FUNCTION_BLOCK MagneticGripper (* Composite FB wrapping other FBs *)
  (* Standard: 61499-2 *)
  (* Version 1.0, 2021-03-18, AK120569 *)
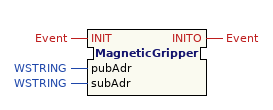
  EVENT_INPUT
    INIT; (* Initialization Request *)
  END_EVENT
  EVENT_OUTPUT
    INITO; (* Initialization Confirm *)
  END_EVENT
  VAR_INPUT
    pubAdr : WSTRING;
    subAdr : WSTRING;
  END_VAR
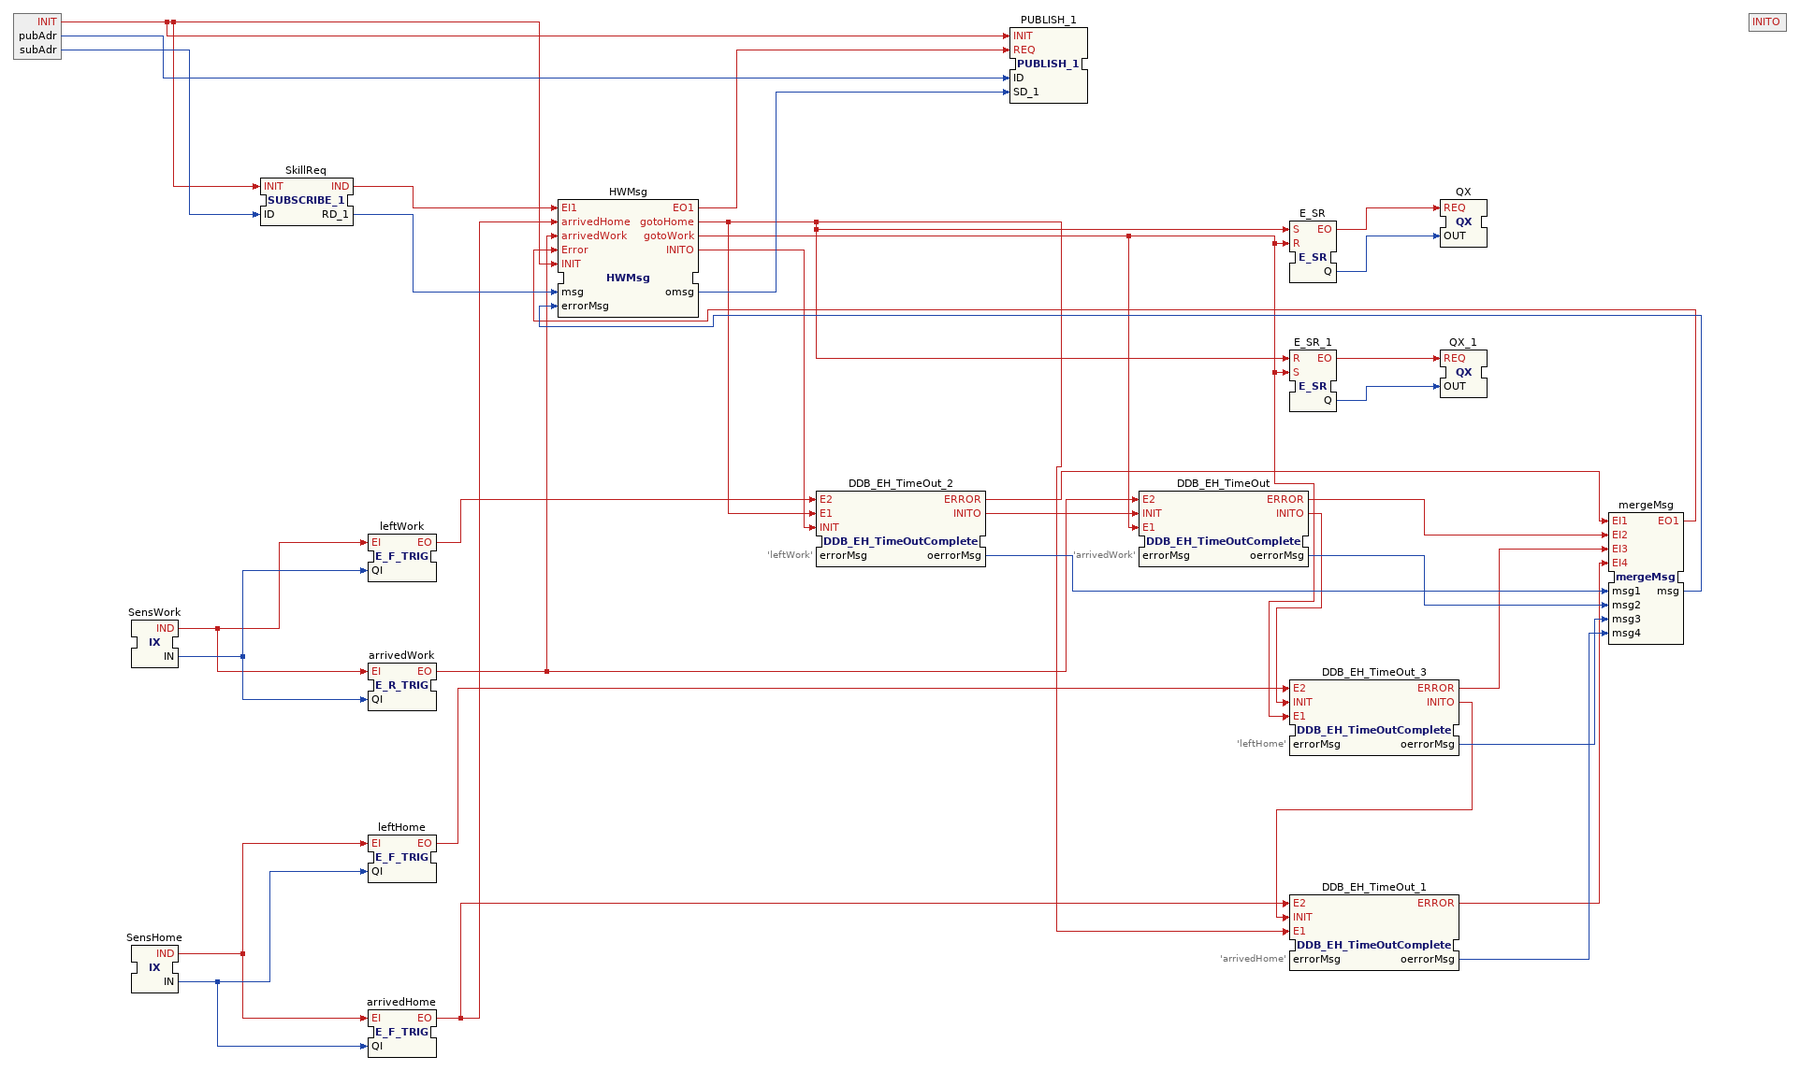
  FBS
    SkillReq : SUBSCRIBE_1;
    SensHome : IX;
    SensWork : IX;
    arrivedHome : E_F_TRIG;
    arrivedWork : E_R_TRIG;
    DDB_EH_TimeOut_1 : DDB_EH_TimeOutComplete(errorMsg := 'arrivedHome');
    DDB_EH_TimeOut : DDB_EH_TimeOutComplete(errorMsg := 'arrivedWork');
    QX : QX;
    QX_1 : QX;
    DDB_EH_TimeOut_2 : DDB_EH_TimeOutComplete(errorMsg := 'leftWork');
    leftWork : E_F_TRIG;
    DDB_EH_TimeOut_3 : DDB_EH_TimeOutComplete(errorMsg := 'leftHome');
    leftHome : E_F_TRIG;
    E_SR : E_SR;
    E_SR_1 : E_SR;
    PUBLISH_1 : PUBLISH_1;
    mergeMsg : mergeMsg;
    HWMsg : HWMsg;
  END_FBS
  EVENT_CONNECTIONS
    SensHome.IND TO arrivedHome.EI;
    SensWork.IND TO arrivedWork.EI;
    arrivedHome.EO TO DDB_EH_TimeOut_1.E2;
    arrivedWork.EO TO DDB_EH_TimeOut.E2;
    SensWork.IND TO leftWork.EI;
    leftWork.EO TO DDB_EH_TimeOut_2.E2;
    SensHome.IND TO leftHome.EI;
    leftHome.EO TO DDB_EH_TimeOut_3.E2;
    E_SR.EO TO QX.REQ;
    E_SR_1.EO TO QX_1.REQ;
    DDB_EH_TimeOut_2.ERROR TO mergeMsg.EI1;
    DDB_EH_TimeOut.ERROR TO mergeMsg.EI2;
    DDB_EH_TimeOut_3.ERROR TO mergeMsg.EI3;
    DDB_EH_TimeOut_1.ERROR TO mergeMsg.EI4;
    INIT TO PUBLISH_1.INIT;
    INIT TO SkillReq.INIT;
    DDB_EH_TimeOut_2.INITO TO DDB_EH_TimeOut.INIT;
    DDB_EH_TimeOut.INITO TO DDB_EH_TimeOut_3.INIT;
    DDB_EH_TimeOut_3.INITO TO DDB_EH_TimeOut_1.INIT;
    SkillReq.IND TO HWMsg.EI1;
    arrivedHome.EO TO HWMsg.arrivedHome;
    arrivedWork.EO TO HWMsg.arrivedWork;
    mergeMsg.EO1 TO HWMsg.Error;
    HWMsg.EO1 TO PUBLISH_1.REQ;
    HWMsg.gotoHome TO DDB_EH_TimeOut_1.E1;
    HWMsg.gotoHome TO DDB_EH_TimeOut_2.E1;
    HWMsg.gotoHome TO E_SR.S;
    HWMsg.gotoHome TO E_SR_1.R;
    HWMsg.gotoWork TO DDB_EH_TimeOut.E1;
    HWMsg.gotoWork TO DDB_EH_TimeOut_3.E1;
    HWMsg.gotoWork TO E_SR.R;
    HWMsg.gotoWork TO E_SR_1.S;
    INIT TO HWMsg.INIT;
    HWMsg.INITO TO DDB_EH_TimeOut_2.INIT;
  END_CONNECTIONS
  DATA_CONNECTIONS
    SensHome.IN TO arrivedHome.QI;
    SensWork.IN TO arrivedWork.QI;
    SensWork.IN TO leftWork.QI;
    SensHome.IN TO leftHome.QI;
    E_SR.Q TO QX.OUT;
    E_SR_1.Q TO QX_1.OUT;
    DDB_EH_TimeOut_2.oerrorMsg TO mergeMsg.msg1;
    DDB_EH_TimeOut.oerrorMsg TO mergeMsg.msg2;
    DDB_EH_TimeOut_3.oerrorMsg TO mergeMsg.msg3;
    DDB_EH_TimeOut_1.oerrorMsg TO mergeMsg.msg4;
    pubAdr TO PUBLISH_1.ID;
    subAdr TO SkillReq.ID;
    SkillReq.RD_1 TO HWMsg.msg;
    mergeMsg.msg TO HWMsg.errorMsg;
    HWMsg.omsg TO PUBLISH_1.SD_1;
  END_CONNECTIONS
END_FUNCTION_BLOCK
